# EPICS substitutions: ek9000App/Db/EL3104.substitutions
file EL3104.template
{       pattern
        {
                TERMINAL,

        }
        {
        }
}
